Fanuc KAREL source: port_GIN.kl

PROGRAM TP
%NOLOCKGROUP
VAR
 x: INTEGER
BEGIN
 x = GIN[3]
END TP
